Staubli VAL3: onLeftEvent.pgx

program onLeftEvent(bool& x_bSave)
  local num i
  local num l_nType
  local string l_sPath
  local string l_sEmpty
  local num l_nResult
  local string l_sMessage
begin
  // left click
  //
  //
  // select the previous one
  //
  if x_bSave
    x_bSave=false
    l_sEmpty=""
    l_nResult=0
    call trajType:onSave(l_sEmpty)
    // show the message
    call language:message(l_sMessage,-4)
    call use:timerDialog(l_sMessage,1)
  endIf
  // check it
  do
    nType=(nType+size(saveData:sTrajType)-1)%(size(saveData:sTrajType))
    saveData:sTrajTypeUsing=saveData:sTrajType[nType]
    if saveData:sTrajType[nType]!=""
      // find the good id
      call saveData:getPathInstr(saveData:sTrajType[nType],l_sPath)
    endIf
  until saveData:sTrajType[nType]!=""
  // load the type
  if trajType:libPath()!=l_sPath and l_sPath!=""
    i=trajType:libLoad(l_sPath)
    delay(0)
  endIf
  if l_sPath==""
    popUpMsg("error load traj type on ENTER "+saveData:sTrajTypeUsing+toString("",i))
  endIf
  // clean the user MENU
  call cleanUserMenu()
  // rebuild the list
  call buildList()
end
